Staubli VAL3: massage.pgx

program massage(string x_sString (dimensions=1))
begin

  call use:clear(0,12)
  gotoxy(0,12)
  put(x_sString)

end
